% RSLogix 500 project LAB06.2.RSS, saved by version 8.30.00.16 %
PROJECT "LAB06.2"    % processor: Bul.1763 MicroLogix 1100 Series B %

PROGRAM FILES
  LAD 2   5 rungs

DATA FILES
  O0 OUTPUT  4 elements
  I1 INPUT  6 elements
  S2 STATUS  66 elements
  B3 BINARY  1 elements
  T4 TIMER  1 elements
  C5 COUNTER  1 elements
  R6 CONTROL  1 elements
  N7 INTEGER  1 elements
  F8 FLOAT  1 elements

LADDER 2
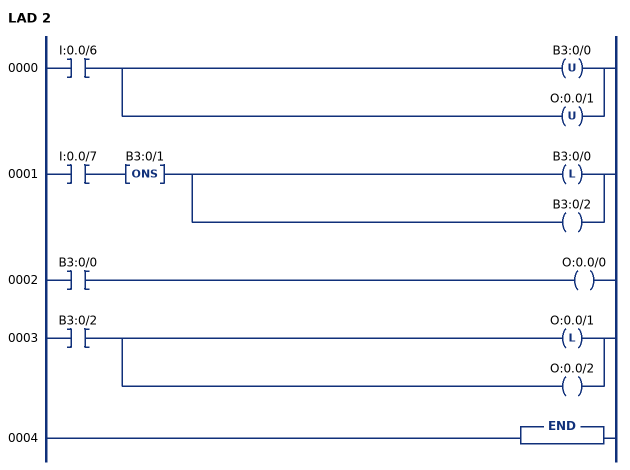
% Rung: 0 %  % edit flag set %
SOR XIC I:0.0/6 BST OTU B3:0/0 NXB OTU O:0.0/1 BND EOR
% Rung: 1 %  % edit flag set %
SOR XIC I:0.0/7 ONS B3:0/1 BST OTL B3:0/0 NXB OTE B3:0/2 BND EOR
% Rung: 2 %  % edit flag set %
SOR XIC B3:0/0 OTE O:0.0/0 EOR
% Rung: 3 %  % edit flag set %
SOR XIC B3:0/2 BST OTL O:0.0/1 NXB OTE O:0.0/2 BND EOR
% Rung: 4 %
SOR END EOR
